FUNCTION_BLOCK FB_SoftStop
VAR_INPUT
	fPosition	 		: LREAL;
	fNormalizedInput 	: LREAL;
	stSoftstop 			: ST_SoftStop;
END_VAR
VAR_OUTPUT
	bSoftStopActive : BOOL;
END_VAR
VAR
END_VAR

IF NOT(stSoftstop.bEnable) THEN
	bSoftStopActive := FALSE;
ELSE
	IF fPosition > stSoftstop.fPosStop AND fNormalizedInput > 0 THEN
		bSoftStopActive := TRUE;
	ELSIF fPosition < stSoftstop.fNegStop AND fNormalizedInput < 0 THEN
		bSoftStopActive := TRUE;
	ELSE
		bSoftStopActive := FALSE;
	END_IF
END_IF

END_FUNCTION_BLOCK

(* stored: Version 1.1.0.1, ProductVersion 3.1.4024.11
   POU FB_SoftStop: Id {8ee418a4-cae3-49ba-96a9-1ad2516d590a}, SpecialFunc None *)
